TYPE stJoint2 :
STRUCT
	left : LREAL;
	right : LREAL;
END_STRUCT
END_TYPE

(* stored: Version 1.1.0.1, ProductVersion 3.1.4026.18
   DUT stJoint2: Id {b1b2c3d4-2222-2222-2222-222222222222} *)
